FUNCTION_BLOCK JOG_CONV
VAR_INPUT
	BOOL_FWD_JOG : BOOL;
	BOOL_RWD_JOG : BOOL;
	UINT_JOG_SPD_MM : UINT;
	TIME_JOG_DELAY : TIME;
	UINT_PLS_RATIO : UINT;

END_VAR
VAR_OUTPUT
	JOG_ACTIVE_BOOL : BOOL;
	JOG_SPD_UINT : UINT;


END_VAR
VAR
	VUINT: UINT;
	T1: TON;
	TI: TIME;
	JSPD_PLS: UINT;
END_VAR
VAR // added by the converter: edge detectors and wires of the graphical bodies
    _w1, _w2 : UINT;
END_VAR

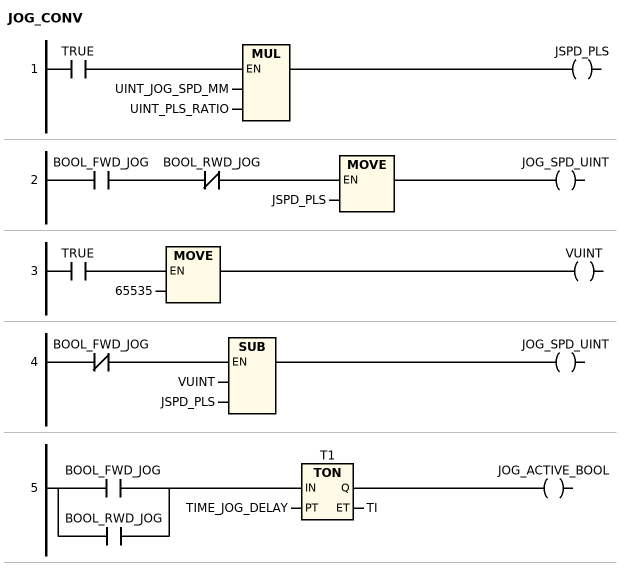
// NETWORK 1
JSPD_PLS := UINT_JOG_SPD_MM * UINT_PLS_RATIO;

// NETWORK 2
IF BOOL_FWD_JOG AND NOT BOOL_RWD_JOG THEN _w1 := JSPD_PLS; END_IF
JOG_SPD_UINT := _w1;

// NETWORK 3
VUINT := 65535;

// NETWORK 4
IF NOT BOOL_FWD_JOG THEN _w2 := VUINT - JSPD_PLS; END_IF
JOG_SPD_UINT := _w2;

// NETWORK 5
T1(IN := BOOL_FWD_JOG OR BOOL_RWD_JOG, PT := TIME_JOG_DELAY, ET => TI); // TON
JOG_ACTIVE_BOOL := T1.Q;

END_FUNCTION_BLOCK

(* stored: Version 1.1.0.1, ProductVersion 3.1.4024.12
   POU JOG_CONV: Id {8766b390-f2cd-49cc-879c-e3503ebadac3}, SpecialFunc None *)
